FUNCTION f_GetISOLvalue : REAL
VAR_INPUT
	rVoltage : REAL;
END_VAR
VAR
	rVoltagePerOhmRate : REAL := 5100/0.889;
END_VAR

f_GetISOLvalue := rVoltage * rVoltagePerOhmRate;

END_FUNCTION

(* stored: Version 1.1.0.1, ProductVersion 3.1.4020.3
   POU f_GetISOLvalue: Id {e05e55c7-3863-4ff6-8853-c8b3df79a4c8}, SpecialFunc None *)
